TYPE ST_System_Calibration :
STRUCT
	Powerstack			: ST_Powerstack_calibration;
END_STRUCT
END_TYPE

(* stored: Version 1.1.0.1, ProductVersion 3.1.4026.18
   DUT ST_System_Calibration: Id {7f4856bf-4a6a-4187-a7a5-0298b7be5b44} *)
